// TIA Portal V17 export
// export: Created 2026-04-13T11:12:45.5164599Z, ExportSetting WithDefaults, DisplayName Totally Integrated Automation Portal, DisplayVersion V17 Update 4, DisplayName TIA Portal Openness, DisplayVersion V17 Update 4, DisplayName TIA Portal Version Control Interface, DisplayVersion V17, DisplayName SINAMICS Startdrive Advanced, DisplayVersion V17, DisplayName SINAMICS Startdrive G130, G150, S120, S150, SINAMICS MV, S210, DisplayVersion V17, DisplayName SINAMICS Startdrive G110M, G120, G120C, G120D, G120P, G115D, DisplayVersion V17, DisplayName STEP 7 Professional, DisplayVersion V17 Update 4, DisplayName STEP 7 Safety, DisplayVersion V17, DisplayName WinCC Professional, DisplayVersion V17 Update 4
VAR_GLOBAL   // PLC tag table "MTX"
   MLS冷水机状态2 AT %MW208 : Int;
   MLS冷水机状态3 AT %MW210 : Int;
   MLS冷水机通信状态 AT %M211.7 : Bool;
   MLS冷水机加热状态 AT %M211.6 : Bool;
   MLS冷水机制冷状态 AT %M211.5 : Bool;
   MLS冷水机超温报警 AT %M209.7 : Bool;
   MLS冷水机低温报警 AT %M209.6 : Bool;
   MLS冷水机压力报警 AT %M209.5 : Bool;
END_VAR
